(* CoDeSys 2.3 project: log-lib-all.pro *)
(* Author: HP *)
(* Libraries: TcBase.lib 14.5.09 12:14:08, TcSystem.lib*7.6.16 11:01:22, TcpIp.lib 6.5.15 08:25:52, STANDARD.LIB 5.6.98 12:03:02 *)

(* Task configuration *)
TASK Standard (PRIORITY := 0, INTERVAL := T#100ms);
	MAIN
END_TASK

(* POU MAIN, ST *)
PROGRAM MAIN
VAR
END_VAR
;
END_PROGRAM
